	FT_PID_0: BURKERT_OSCAT_BASIC.CTRL_PID;
	GEN_PULSE_0: BURKERT_OSCAT_BASIC.GEN_PULSE;
	In_Zone: BOOL;
	TON_0: TON;
	R_TRIG_0: R_trig;
	Timer_Status: INT;
	ABS_Error: REAL;
	R_TRIG_1: R_trig;
	RAMP_REAL_0: Util.RAMP_REAL;
	SR_0: SR;
	TON_1: TON;
	TOF_0: TOF;
	TON_2: TON;
	FT_PID_1:Util.PID_FIXCYCLE;
	
	R_trig_2:R_Trig;
	Loop_Disable:BOOL;
	TP_1:TP;
	
	FT_PIDWL_0: BURKERT_OSCAT_BASIC.FT_PIDWL;
	FT_PIDW_0: BURKERT_OSCAT_BASIC.FT_PIDW;
	TOF_1: TOF;
	On_Seconds: REAL;
	PID_Reset: BOOL;
	TON_3: TON;
	TP_0: TP;
	Current_Minute: UINT;
	R_TRIG_3: R_trig;
	TON_4: TON;
	Profile_Reset: BOOL;
END_VAR
VAR_OUTPUT

END_VAR
VAR // added by the converter: edge detectors and wires of the graphical bodies
    _w1, _w2, _w3, _w4, _w7, _w8, _w10, _w12, _w13, _w14, _w15, _w19, _w21, _w23, _w25, _w27 : ANY;
    _w5, _w11 : TIME;
    _w6, _w9, _w16, _w17, _w18, _w20, _w22, _w24, _w26 : BOOL;
END_VAR

// note: 7 stored wires end on pins the file does not list and are not shown
BCV_Loop.DeadBand := SEL(BCV_Loop.DeadBand = 0.0, BCV_Loop.DeadBand, 0.1);
BCV_Loop.Live_Target_EU := SEL(BCV_Loop.Mode=Temp_Loop_Modes.Step, BCV_Loop.Target_EU, SEL(HEATING, TT.EU-(BCV_Loop.DeadBand*1.5), TT.EU+(BCV_Loop.DeadBand*1.5)));
_w1 := (BCV_Loop.Mode = Temp_Loop_Modes.Crash) OR (BCV_Loop.Mode = Temp_Loop_Modes.Step);
_w2 := ABS(BCV_Loop.Target_EU - TT.EU);
ABS_Error := _w2;
(* _w2 * BCV_Loop.kp < 50; result not used *)
TON_2(IN := False OR _w2 < BCV_Loop.Window, PT := T#5s); // TON
_w3 := _w1 AND TON_2.Q;
In_Zone := _w3;
R_TRIG_0(CLK := _w1 AND _w3); // R_trig
IF R_TRIG_0.Q THEN _w4 := Temp_Loop_Modes.Auto; END_IF
BCV_Loop.Mode := _w4;
_w5 := REAL_TO_TIME(BCV_LOOP.Min_Cycle_S) * 1000;
_w6 := On_Seconds > BCV_LOOP.Min_Cycle_S;
_w7 := SEL(Heating, BCV_Loop.Live_Target_EU, BCV_Loop.Actual_EU);
_w8 := SEL(Heating, BCV_Loop.Actual_EU, BCV_Loop.Live_Target_EU);
TOF_0(IN := Permisive, PT := T#15s); // TOF
TON_3(IN := TOF_0.Q, PT := T#15s); // TON
_w9 := On_Seconds > BCV_LOOP.Max_Cycle_S - BCV_LOOP.Min_Cycle_S;
SR_0(SET1 := Loop_Disable, RESET := BCV_Loop.Mode=Temp_Loop_Modes.Idle); // SR
TP_1(IN := _w3, PT := T#5s); // TP
IF SR_0.Q1 THEN _w10 := Temp_Loop_Modes.Idle; END_IF
BCV_Loop.Mode := _w10;
_w11 := UINT_TO_TIME(BCV_Loop.Timer_Target_M) * 60000;
TOF_1(IN := (TT.Status.eStatus=Burkert.eSensor_Status.Offline) OR (TT.Status.eStatus=Burkert.eSensor_Status.Fault), PT := t#15s); // TOF
_w12 := (BCV_Loop.Mode=Temp_Loop_Modes.Auto_Paused) OR (BCV_Loop.Mode=Temp_Loop_Modes.Idle) OR NOT TON_3.Q OR SR_0.Q1 OR (BCV_Loop.Status=Temp_Loop_Status.Timer_Expired) OR TOF_1.Q;
_w13 := _w12 OR (_w12 OR TP_1.Q);
PID_Reset := _w13;
FT_PIDW_0(
    IN := SEL(_w12, _w8, _w7) - _w7,
    KP := BCV_Loop.kp,
    TN := BCV_Loop.TN,
    TV := BCV_Loop.TV,
    LIM_L := 0,
    LIM_H := 100,
    RST := _w13); // BURKERT_OSCAT_BASIC.FT_PIDW
BCV_Loop.Limiter := FT_PIDW_0.LIM;
_w14 := SEL(PID_Reset, SEL(BCV_Loop.Mode=Temp_Loop_Modes.Crash, FT_PIDW_0.Y, 100.0), 0.0);
BCV_Loop.Load_EU := _w14;
_w15 := _w14 * ((BCV_Loop.Max_Cycle_S/100.0));
On_Seconds := _w15;
GEN_PULSE_0(
    ENQ := _w6,
    PTH := REAL_TO_TIME(_w15) * 1000,
    PTL := REAL_TO_TIME(BCV_LOOP.Max_Cycle_S - _w15) * 1000); // BURKERT_OSCAT_BASIC.GEN_PULSE
_w16 := _w6 AND GEN_PULSE_0.Q;
TP_0(IN := _w16, PT := _w5); // TP
_w17 := (TP_0.Q OR _w16 OR _w9) AND NOT Loop_Disable AND NOT (BCV_Loop.Mode=Temp_Loop_Modes.Idle);
BCV_Loop.Output := _w17;
BCV.PLC_CMD := _w17;
_w18 := (BCV_Loop.Mode=Temp_Loop_Modes.Profile) AND (BCV_Loop.Timer_Target_M>0) AND NOT _w13 AND NOT Profile_Reset;
TON_0(IN := _w18, PT := _w11); // TON
Current_Minute := TIME_TO_UINT(TON_0.ET / 60000);
BCV_Loop.Timer_Remaining_s := TIME_TO_UINT((_w11 - TON_0.ET) / 1000);
TT.Burkert.cAlarm_Config.Hi_Hi_Alarm := SEL(NOT _w12, TT.Burkert.cAlarm_Config.Hi_Hi_Alarm, BCV_Loop.Live_Target_EU+(BCV_Loop.Window*2));
_w19 := (TT.Status.eStatus=Burkert.eSensor_Status.Offline) OR (TT.Status.eStatus=Burkert.eSensor_Status.Offline);
Loop_Disable := External_Fault OR (TT.Status.eStatus=Burkert.eSensor_Status.FORCED) OR (BCV.Mode<>eBCV_Modes.Auto) OR _w19;
TT.Burkert.cAlarm_Config.Hi_Warn := SEL(NOT _w12, TT.Burkert.cAlarm_Config.Hi_Warn, BCV_Loop.Live_Target_EU+(BCV_Loop.Window));
TT.Burkert.cAlarm_Config.Low_warn := SEL(NOT _w12, TT.Burkert.cAlarm_Config.Low_warn, BCV_Loop.Live_Target_EU-(BCV_Loop.Window));
TT.Burkert.cAlarm_Config.Low_Low_Alarm := SEL(NOT _w12, TT.Burkert.cAlarm_Config.Low_Low_Alarm, BCV_Loop.Live_Target_EU-(BCV_Loop.Window*2));
BCV_Loop.Status := SEL(BCV.Mode<>eBCV_Modes.Auto, SEL(TT.Status.eStatus=Burkert.eSensor_Status.FORCED, SEL(External_Fault, SEL(_w19, SEL(BCV_Loop.Mode=Temp_Loop_Modes.Auto_Paused, SEL(BCV_Loop.Mode=Temp_Loop_Modes.Idle, SEL(TT.Status.eStatus=Burkert.eSensor_Status.Low_Low_Alarm, SEL(TT.Status.eStatus=Burkert.eSensor_Status.Low_Warning, SEL(TT.Status.eStatus=Burkert.eSensor_Status.HiHi_Alarm, SEL(TT.Status.eStatus=Burkert.eSensor_Status.High_Warning, SEL(TON_0.Q, SEL(_w18, SEL(BCV_Loop.Mode=Temp_Loop_Modes.Auto, SEL(Permisive, Temp_Loop_Status.Pre_Start, Temp_Loop_Status.Ramping), Temp_Loop_Status.Auto), Temp_Loop_Status.Timed), Temp_Loop_Status.Timer_Expired), Temp_Loop_Status.HiHi_Warning), Temp_Loop_Status.HiHi_Alarm), Temp_Loop_Status.LoLo_Warning), Temp_Loop_Status.LoLo_Alarm), Temp_Loop_Status.Idle), Temp_Loop_Status.Paused), Temp_Loop_Status.Fault), Temp_Loop_Status.External_Fault), Temp_Loop_Status.Sensor_Forced), Temp_Loop_Status.Valve_Not_auto);
BCV_Loop.Actual_EU := TT.EU;
BCV_Loop.Error_EU := SEL(BCV_Loop.Mode=Temp_Loop_Modes.Idle, TT.EU - BCV_Loop.Target_EU, 0.0);
BCV_Loop.Int_Out := FT_PIDW_0.YI;
BCV_Loop.Diff_Out := FT_PIDW_0.diff.out;
TT.Alarm_Config.Silence := BCV_Loop.Mode=Temp_Loop_Modes.Idle;
R_TRIG_3(CLK := BCV_Loop.Mode=Temp_Loop_Modes.Profile); // R_trig
_w20 := R_TRIG_3.Q;
IF _w20 THEN _w21 := 0; END_IF
BCV_Loop.Temp_Profile.Index := _w21;
_w22 := (BCV_Loop.Mode=Temp_Loop_Modes.Profile) AND (BCV_Loop.Timer_Remaining_s=1) AND NOT (BCV_Loop.Temp_Profile.Index=4);
IF _w22 THEN _w23 := BCV_Loop.Temp_Profile.Index+1; END_IF
BCV_Loop.Temp_Profile.Index := _w23;
_w24 := (_w20 OR _w22) AND NOT (BCV_Loop.Temp_Profile.Time_m[BCV_Loop.Temp_Profile.Index]=0);
IF _w24 THEN _w25 := BCV_Loop.Temp_Profile.Time_m[BCV_Loop.Temp_Profile.Index]; END_IF
BCV_Loop.Timer_Target_M := _w25;
_w26 := _w24;
IF _w26 THEN _w27 := BCV_Loop.Temp_Profile.Target[BCV_Loop.Temp_Profile.Index]; END_IF
Profile_Reset := _w26;
BCV_Loop.Target_EU := _w27;
// TRUE: input not connected
// Temp_Loop_Status.Idle: input not connected

END_FUNCTION_BLOCK

// Chase_Master_Rate_UDFB
FUNCTION_BLOCK Chase_Master_Rate_UDFB
VAR_INPUT
	Valve_Ready:BOOL;
	Valve_Open:Bool;
END_VAR
VAR_OUTPUT
	BCV_CMD:BOOL;
	ACV_CMD:REAL;
END_VAR
VAR
	Run_Request:Bool;
	
END_VAR
VAR_IN_OUT
	chase:cChase;
	FIT:Burkert.cFIT;
	Flow_PID:PID_DUT;
	//Temp_PID:PID_DUT;
END_VAR

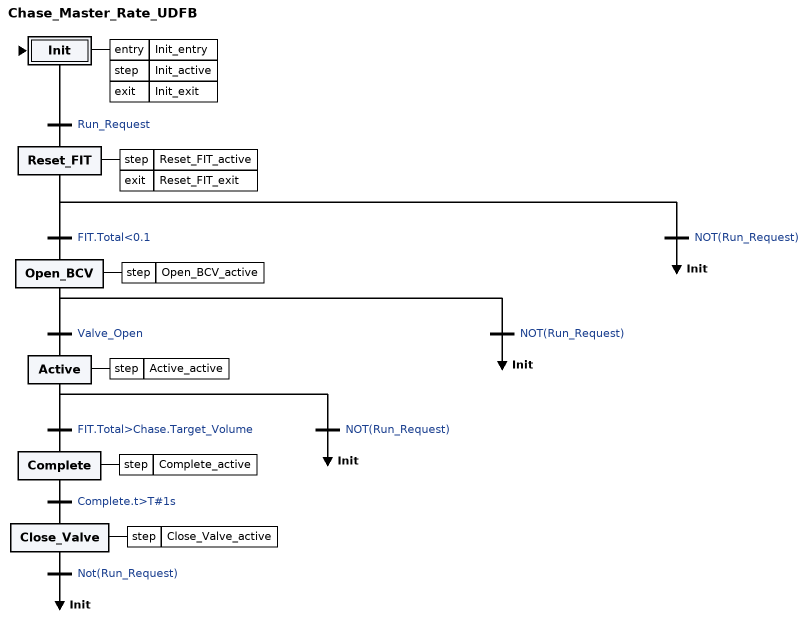
INITIAL_STEP Init:
    Init_entry(P1);  // entry action
    Init_active(N);  // step action
    Init_exit(P0);  // exit action
END_STEP
TRANSITION FROM Init TO Reset_FIT
    := Run_Request;
END_TRANSITION
STEP Reset_FIT:
    Reset_FIT_active(N);  // step action
    Reset_FIT_exit(P0);  // exit action
END_STEP
TRANSITION FROM Reset_FIT TO Open_BCV
    := FIT.Total<0.1;
END_TRANSITION
STEP Open_BCV:
    Open_BCV_active(N);  // step action
END_STEP
TRANSITION FROM Open_BCV TO Active
    := Valve_Open;
END_TRANSITION
TRANSITION FROM Open_BCV TO Init
    := NOT(Run_Request);
END_TRANSITION
STEP Active:
    Active_active(N);  // step action
END_STEP
TRANSITION FROM Active TO Complete
    := FIT.Total>Chase.Target_Volume;
END_TRANSITION
TRANSITION FROM Active TO Init
    := NOT(Run_Request);
END_TRANSITION
STEP Complete:
    Complete_active(N);  // step action
END_STEP
TRANSITION FROM Complete TO Close_Valve
    := Complete.t>T#1s;
END_TRANSITION
STEP Close_Valve:
    Close_Valve_active(N);  // step action
END_STEP
TRANSITION FROM Close_Valve TO Init
    := Not(Run_Request);
END_TRANSITION
TRANSITION FROM Reset_FIT TO Init
    := NOT(Run_Request);
END_TRANSITION

END_FUNCTION_BLOCK

// Chase_Master_UDFB
FUNCTION_BLOCK Chase_Master_UDFB
VAR_INPUT
	Valve_Ready:BOOL;
END_VAR
VAR_OUTPUT
	BCV_CMD:BOOL;
	ACV_CMD:REAL;
END_VAR
VAR
	Run_Request:Bool;
	
END_VAR
VAR_IN_OUT
	chase:cChase;
	FIT:Burkert.cFIT;
	Flow_PID:PID_DUT;
	Temp_PID:PID_DUT;
END_VAR

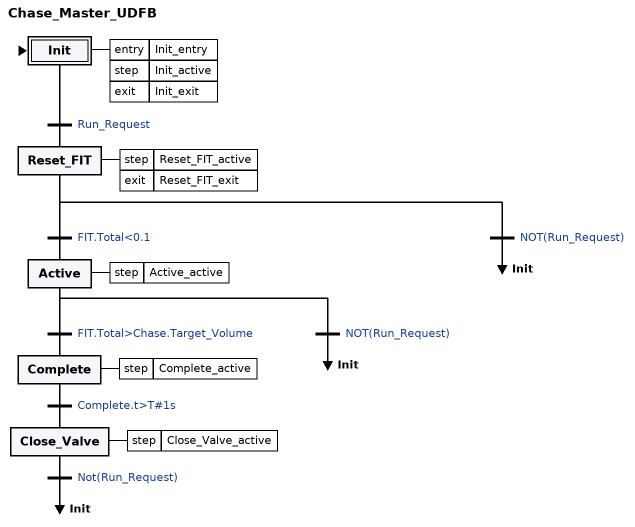
INITIAL_STEP Init:
    Init_entry(P1);  // entry action
    Init_active(N);  // step action
    Init_exit(P0);  // exit action
END_STEP
TRANSITION FROM Init TO Reset_FIT
    := Run_Request;
END_TRANSITION
STEP Reset_FIT:
    Reset_FIT_active(N);  // step action
    Reset_FIT_exit(P0);  // exit action
END_STEP
TRANSITION FROM Reset_FIT TO Active
    := FIT.Total<0.1;
END_TRANSITION
STEP Active:
    Active_active(N);  // step action
END_STEP
TRANSITION FROM Active TO Complete
    := FIT.Total>Chase.Target_Volume;
END_TRANSITION
TRANSITION FROM Active TO Init
    := NOT(Run_Request);
END_TRANSITION
STEP Complete:
    Complete_active(N);  // step action
END_STEP
TRANSITION FROM Complete TO Close_Valve
    := Complete.t>T#1s;
END_TRANSITION
STEP Close_Valve:
    Close_Valve_active(N);  // step action
END_STEP
TRANSITION FROM Close_Valve TO Init
    := Not(Run_Request);
END_TRANSITION
TRANSITION FROM Reset_FIT TO Init
    := NOT(Run_Request);
END_TRANSITION

END_FUNCTION_BLOCK

// Chase_Slave_UDFB
FUNCTION_BLOCK Chase_Slave_UDFB
VAR_INPUT
	Source_Healthy:BOOL;
	Destination_Healthy:BOOL;
	
END_VAR
VAR_OUTPUT
	BCV_CMD:BOOL;
END_VAR
VAR
	Chase_Request:BOOL;
END_VAR
VAR_IN_OUT
	Transfer:cChase;
	Chase:cChase;
END_VAR

Chase_Request:= (Chase.Mode=eChase_Mode.Auto AND Chase.PLC_Run) OR Chase.Mode=eChase_mode.Manual;
IF (Transfer.Status.eStatus=Transfer_Status.IDLE  AND Chase_Request) THEN
	Chase.Active:=TRUE;
END_IF;


IF (Transfer.Status.eStatus=Transfer_Status.IDLE AND Source_Healthy AND Destination_Healthy AND Chase_Request) OR Chase.Active THEN
	Transfer.Mode:=Chase.Mode;
	Transfer.PLC_Run:=Chase.PLC_Run;
	Transfer.Target_Rate:=Chase.Target_Rate;
	Transfer.Target_Temp:=Chase.Target_Temp;
	Transfer.Target_Volume:=Chase.Target_Volume;
	//Chase.Active:=Transfer.Active;
	Chase.Status.eStatus:=Transfer.Status.eStatus;
	Chase.PCT_Remain:=Transfer.PCT_Remain;
	Chase.ETA:=Transfer.ETA;
	BCV_CMD:=(Transfer.Status.eStatus=eChase_Status.Active);
	
ELSE
	//Chase.Active:=FALSE;
	BCV_CMD:=FALSE;
	IF NOT(Destination_Healthy) THEN
		Chase.Status.eStatus:=eChase_Status.Destination_Not_Ready;
	END_IF;
	IF NOT(Source_Healthy) THEN
		Chase.Status.eStatus:=eChase_Status.Source_Not_Ready;
	END_IF;
	IF (Transfer.Status.eStatus<>Transfer_Status.IDLE) THEN
		Chase.Status.eStatus:=eChase_Status.Not_Available;
	END_IF;
	
END_IF;

IF Chase.Active AND NOT(Chase_request) THEN
		Transfer.Mode:=Chase.Mode;
		Transfer.PLC_Run:=Chase.PLC_Run;
		Chase.Active:=FALSE;
END_IF

IF(Chase.Status.eStatus=eChase_Status.Not_Available AND Transfer.Status.eStatus=eChase_Status.IDLE) THEN
	Chase.Status.eStatus:=Transfer.Status.eStatus;
END_IF;
IF(Chase.Status.eStatus=eChase_Status.Source_Not_Ready AND Source_Healthy) THEN
	Chase.Status.eStatus:=eChase_Status.IDLE;
END_IF;
IF(Chase.Status.eStatus=eChase_Status.Destination_Not_Ready AND Destination_Healthy) THEN
	Chase.Status.eStatus:=eChase_Status.IDLE;
END_IF;

END_FUNCTION_BLOCK

// PLC_TIME
{attribute 'hide_all_locals’}
PROGRAM PLC_TIME
VAR_INPUT
(* Change PLC Time *)
    (* User command for updating the controller's date & time *)
    i_xCmdSetDateTime           : BOOL  := FALSE;
    (* New Date: Date & Time elements for a SYSTEMDATE structure *)
    i_uiYear                    : UINT  := 2011; 
    i_uiMonth                   : UINT  :=    1; (* Mounths 1 to 12 *)
    i_uiDay                     : UINT  :=    1; (* Days 1 to 31 *)
    i_uiHour                    : UINT  :=   11; (* Hours 0 to 23 *)
    i_uiMinutes                 : UINT  :=   55; (* Minutes 0 to 59 *)
    i_uiSeconds                 : UINT  :=    0; (* Seconds 0 to 59 *)
	i_diMinuntesOffset			: DINT	:= 0; //Time Offset from UTC	
END_VAR
VAR_OUTPUT
	q_uiYear                    : UINT  := 0;
    q_uiMonth                   : UINT  := 0;
    q_uiDay                     : UINT  := 0;
    q_uiHour                    : UINT  := 0;
    q_uiMinutes                 : UINT  := 0;
    q_uiSeconds                 : UINT  := 0;
    q_uiDayOfWeek               : UINT  := 0;
    q_uiDayOfYear               : UINT  := 0;
	q_dwEpochTime				: DWORD;	
END_VAR

VAR
	(* Read PLC Time *)
    (* Result: Controller RTC as a UTC Timestamp value      *)
    (* (number of seconds since January 1st, 1970 00:00:00) *)
	{attribute 'symbol' := 'none'}
    v_dwControllerRtcAsUtc      : DWORD := 0;
    (* Result: Date & Time in a SYSTEMDATE structure *)
	{attribute 'symbol' := 'none'}
    v_PLCDate                   : SYSTIMEDATE;
    (* Result: Date & Time elements of the SYSTEMDATE structure *)
	    (* Function operation diagnostic of the "SysTimeRtcGet" function: OK if 0 *)
	{attribute 'symbol' := 'none'}
    q_udiSysTimeRtcGetDiag      : UDINT := 0;
    (* Function operation diagnostic of the "SysTimeRtcConvertUtcToDate" function: OK if 0 *)
	{attribute 'symbol' := 'none'}
    q_udiConvertUtcToDateDiag   : UDINT := 0;
(* Change PLC Time *)
    (* New Date: Date & Time as a SYSTEMDATE structure *)
	{attribute 'symbol' := 'none'}
    v_NewPLCDate                : SYSTIMEDATE;
    (* New Date: Timestamp calculated from entered Date & Time value *)
    (*  = number of seconds since January 1st, 1970 00:00:00         *)
    (*    or FFFF FFFF hex in case of unsuccessful conversion.       *)
	{attribute 'symbol' := 'none'}
    v_dwNewControllerRtcAsUtc   : DWORD := 0;
    (* Command for updating the controller's date & time: Only if they are valid *)
	{attribute 'symbol' := 'none'}
    v_xSetValidDateTime         : BOOL  := FALSE;
    (* Function operation diagnostic of the "SysTimeRtcConvertDateToUtc" function: OK if 0 *)
	{attribute 'symbol' := 'none'}
    q_udiConvertDateToUtcDiag   : UDINT := 0;
    (* Function operation diagnostic of the "SysTimeRtcSet" function: OK if 0 *)
	{attribute 'symbol' := 'none'}
    q_udiSysTimeRtcSetDiag      : UDINT := 0;
	i_diMinuntesOffset_test: DINT;
END_VAR

(*****************)
(* Read PLC Time *)
(*****************)

(* IN/OUT - Function operation diagnostic (0 if OK) *)
(* Result = Controller RTC as a UTC Timestamp value (number of seconds since January 1st, 1970 00:00:00) *)
q_dwEpochTime := SysTimeRtcGet(pResult := q_udiSysTimeRtcGetDiag);
q_dwEpochTime := DINT_TO_DWORD(DWORD_TO_DINT(q_dwEpochTime)+i_diMinuntesOffset*60);	

(* IN     - UTC Timestamp value (number of seconds since January 1st, 1970 00:00:00) *)
(* IN/OUT - Date & Time in a SYSTEMDATE structure *)
(* Result = Function operation diagnostic (OK if 0) *)
q_udiConvertUtcToDateDiag := SysTimeRtcConvertUtcToDate(dwTimestampUtc := q_dwEpochTime,  pDate:= v_PLCDate);


(* Date & Time elements of the SYSTEMDATE structure *)
(* Examples of access to any SYSTIMEDATE data: v_PLCDate => v_PLCDate.wXXXXX *)
q_uiYear        := v_PLCDate.wYear;
q_uiMonth       := v_PLCDate.wMonth;
q_uiDay         := v_PLCDate.wDay;
q_uiHour        := v_PLCDate.wHour;
q_uiMinutes     := v_PLCDate.wMinute;
q_uiSeconds     := v_PLCDate.wSecond;
q_uiDayOfWeek   := v_PLCDate.wDayOfWeek;
q_uiDayOfYear   := v_PLCDate.wYday;

(*******************)
(* Change PLC Time *)
(*******************)

(* Date & Time elements for a SYSTEMDATE structure *)
(* NOTE: The "Day of Week" and "Day of Year" elements are not useful here. *)
(* Examples of access to any SYSTIMEDATE data: v_NewPLCDate => v_NewPLCDate.wXXXXX *)
v_NewPLCDate.wYear         := i_uiYear;
v_NewPLCDate.wMonth        := i_uiMonth;
v_NewPLCDate.wDay          := i_uiDay;
v_NewPLCDate.wHour         := i_uiHour;
v_NewPLCDate.wMinute       := i_uiMinutes;
v_NewPLCDate.wSecond       := i_uiSeconds;
v_NewPLCDate.wMilliseconds := 0;

(* IN/OUT - Date & Time as a SYSTEMDATE structure *)
(* IN/OUT - New Date: Timestamp calculated from entered Date & Time value *)
(*           =  number of seconds since January 1st, 1970 00:00:00        *)
(*              or FFFF FFFF hex in case of unsuccessful conversion.      *)
(* Result = Function operation diagnostic (OK if 0) *)
q_udiConvertDateToUtcDiag := SysTimeRtcConvertDateToUtc(pDate:= v_NewPLCDate, pdwTimestampUtc := v_dwNewControllerRtcAsUtc);
v_dwNewControllerRtcAsUtc :=DINT_TO_DWORD(DWORD_TO_DINT(v_dwNewControllerRtcAsUtc)-i_diMinuntesOffset*60);

(* Command for updating the controller's date & time:            *)
(* Only if they are valid AND if in presence of the user command *)
v_xSetValidDateTime := (v_dwNewControllerRtcAsUtc <> 16#FFFFFFFF) AND i_xCmdSetDateTime;

IF v_xSetValidDateTime THEN
    (* IN     - Timestamp of the New Date (number of seconds since January 1st, 1970 00:00:00) *)
    (* Result = Function operation diagnostic (OK if 0) *)
    q_udiSysTimeRtcSetDiag := SysTimeRtcSet(ulTimestamp := v_dwNewControllerRtcAsUtc);
END_IF
i_xCmdSetDateTime:=FALSE;

END_PROGRAM

// Tempered_Mix_eDip_UDFB
FUNCTION_BLOCK Tempered_Mix_eDip_UDFB
VAR_INPUT
	//Loop_ID:INT;
END_VAR
VAR_IN_OUT
	HW_ACV:eDip_8694_DUT;
	CW_ACV:eDip_8694_DUT;
	Temperature:AIT_DUT;
	FIT:FIT_DUT;
	Control:Mix_DUT;
END_VAR
VAR_OUTPUT
END_VAR
VAR
	R_TRIG_0: R_Trig;
	RATE_PID: BURKERT_OSCAT_BASIC.CTRL_PID;
	
	Temp_PID: BURKERT_OSCAT_BASIC.CTRL_PID;
	TON_0: TON;
	Stage_Delay: TIME := T#2s;
	TON_1: TON;
	TON_2: TON;
	SRAMP_0: BURKERT_OSCAT_BASIC.SRAMP;
	TON_3: TON;
	TON_4: TON;
	Ramp_Active: BOOL;
	Ramp_Target: REAL;
	TON_5: TON;
	TON_6: TON;
	R_TRIG_1: R_trig;
	Ramp_Start_Volume: REAL;
	Ramp_Volume: REAL;
	R_TRIG_2: R_Trig;
	R_TRIG_3: R_Trig;
	PID_0: Util.PID;
	R_TRIG_4: R_Trig;
	R_TRIG_5:R_trig;
	Live_Rate:Real;
	
END_VAR
VAR // added by the converter: edge detectors and wires of the graphical bodies
    _w1, _w2, _w3, _w4, _w5, _w6, _w11, _w13, _w14, _w15, _w16, _w17, _w19, _w20, _w23, _w25, _w27, _w33, _w34, _w35, _w37 : ANY;
    _w7, _w8, _w9, _w10, _w12, _w18, _w21, _w22, _w24, _w26, _w28, _w30, _w31, _w32, _w36, _w38 : BOOL;
    _w29 : REAL;
END_VAR

